// TwinCAT 3 PLC project Nepionic_Metrics
// Title: Nepionic_Metrics
// Company: Nepionic
// Author: Nepionic
// ProjectVersion: 0.1.0
// ProgramVersion: 3.1.4026.22
// project tree:
//   Api/ MetricCore.TcIO
//   Lib/ MetricKind.TcDUT, MetricAttribute.TcDUT, Meter.TcPOU

// ---- Lib/MetricKind.TcDUT
{attribute 'qualified_only'}
{attribute 'strict'}
{attribute 'to_string'}
TYPE MetricKind : (
	Gauge := 0,
	Counter := 1,
	UpDownCounter := 2
) UDINT;
END_TYPE

// ---- Lib/MetricAttribute.TcDUT
// A single structured metric attribute — a key/value label attached to a metric data point.
TYPE MetricAttribute :
STRUCT
	key : STRING(31);
	value : STRING(63);
END_STRUCT
END_TYPE

// ---- Api/MetricCore.TcIO
INTERFACE MetricCore

// Record a single metric data point.
// Backends that do not support structured attributes should ignore attrs/attr_count.
METHOD PUBLIC Record : BOOL
VAR_INPUT
	name : STRING(127);
	unit : STRING(31);
	value : LREAL;
	kind : MetricKind;
	attrs : ARRAY[0..4] OF MetricAttribute;
	attr_count : USINT;
END_VAR
END_METHOD

END_INTERFACE

// ---- Lib/Meter.TcPOU
{attribute 'linkalways'}
{attribute 'no_explicit_call' := 'This FB is a CLASS and must be accessed using methods or properties'}
{attribute 'enable_dynamic_creation'}
/// Otel-like metrics client. Wire a MetricCore backend via the Core property,
/// then call Gauge/Counter/UpDownCounter to record data points.
/// Attributes can be attached to the next call using WithAttribute chaining.
///
/// Example:
///   meter.WithAttribute('axis.id', '3').Gauge('plc.axis.position', 'mm', pos);
FUNCTION_BLOCK PUBLIC Meter
VAR
	_core : MetricCore;
	attrs : ARRAY[0..4] OF MetricAttribute;
	attr_count  : USINT;
	initialised : BOOL;
END_VAR

{attribute 'monitoring' := 'call'}
PROPERTY PUBLIC Core : MetricCore
GET // PUBLIC
Core := _core;
END_GET
SET // PUBLIC
_core := Core;
END_SET
END_PROPERTY

/// Record a monotonically increasing counter data point.
METHOD PUBLIC Counter
VAR_INPUT
	name : STRING(127);
	unit : STRING(31);
	value : LREAL;
END_VAR
IF _core <> 0 THEN
	_core.Record(name, unit, value, MetricKind.Counter, attrs, attr_count);
END_IF
attr_count := 0;
initialised := FALSE;
END_METHOD

/// Record a gauge (instantaneous) data point.
METHOD PUBLIC Gauge
VAR_INPUT
	name : STRING(127);
	unit : STRING(31);
	value : LREAL;
END_VAR
IF _core <> 0 THEN
	_core.Record(name, unit, value, MetricKind.Gauge, attrs, attr_count);
END_IF
attr_count := 0;
initialised := FALSE;
END_METHOD

/// Record an up/down counter data point (can increase or decrease).
METHOD PUBLIC UpDownCounter
VAR_INPUT
	name : STRING(127);
	unit : STRING(31);
	value : LREAL;
END_VAR
IF _core <> 0 THEN
	_core.Record(name, unit, value, MetricKind.UpDownCounter, attrs, attr_count);
END_IF
attr_count := 0;
initialised := FALSE;
END_METHOD

/// Attach a key/value attribute to the next metric call. Up to 5 attributes;
/// extras are silently ignored. Resets after each sink call.
METHOD PUBLIC WithAttribute : REFERENCE TO Meter
VAR_INPUT
	key : STRING(31);
	value : STRING(63);
END_VAR
IF NOT initialised THEN
	attr_count := 0;
	initialised := TRUE;
END_IF

IF attr_count < 5 THEN
	attrs[attr_count].key   := key;
	attrs[attr_count].value := value;
	attr_count := attr_count + 1;
END_IF

WithAttribute REF= THIS^;
END_METHOD

END_FUNCTION_BLOCK
